TYPE ST_JXCE1_RxPDO :
STRUCT
	OutputPortSignalsAreAllocated	: WORD;
	NumericalDataFlag				: WORD;
	StartFlag                       : BYTE;
	MovementMode                    : BYTE;
	Speed                           : WORD;
	TargetPosition                  : DINT;
	Acceleration                    : WORD;
	Deceleration                    : WORD;
	PushingForce                    : WORD;
	TriggerLV                       : WORD;
	PushingSpeed                    : WORD;
	MovingForce                     : WORD;
	Area1                           : DINT;
	Area2                           : DINT;
	InPosition                      : DINT;
END_STRUCT
END_TYPE

(* stored: Version 1.1.0.1, ProductVersion 3.1.4024.15
   DUT ST_JXCE1_RxPDO: Id {ccdbac40-c2c0-0561-201d-dcfa7df96a40} *)
